DATA_BLOCK "ALM_DB"
{ S7_Optimized_Access := 'TRUE' }
VERSION : 0.1
NON_RETAIN
   VAR
      // 模拟量报警信息数组[1..40]
      Ana_ALM : Array[1..40] of "UDT_Ana_ALM";

      // 设备控制报警信息数组[1..10]
      Device_ALM : Array[1..10] of "UDT_Device_ALM";

      // 阀门控制报警信息数组[1..15]
      Valve_ALM : Array[1..15] of "UDT_Valve_ALM";
   END_VAR


BEGIN
END_DATA_BLOCK